Universal Robots PolyScope program: David.urp

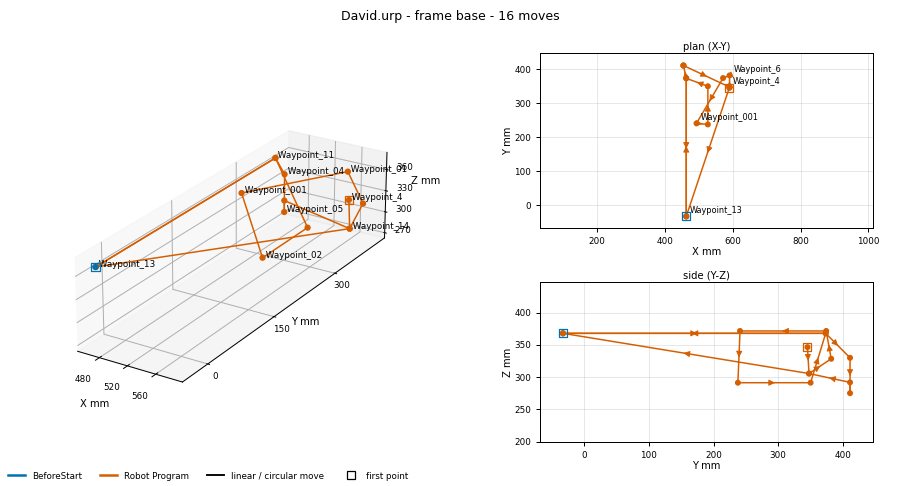
[picture p0: tool path of David.urp in frame base, 16 of 16 moves have a stored position in this frame; points joined in program order, loops and branches not executed]
Program David (installation=robINST_del2David directory=/programs/seminar/2526/zindovic_main createdIn=5.8.0.10253 lastSavedIn=5.8.0.10253 robotSerialNumber=20185500087)
Calibrated DH parameters: a=[0.000137, -0.413209, -0.387078, 0.000078, -0.000004, 0]; d=[0.162361, 46.755621, 39.772032, -86.394282, 0.099723, 0.099655]; alpha=[1.570462, -0.002125, 0.000722, 1.570578, -1.570334, 0]; deltaTheta=[0, -0.236012, 6.679269, -0.160076, 0, 0]
BeforeStart
  MoveJ speed 60 deg/s, acceleration 80 deg/s^2 (useActiveTCP=true) feature=Base
    Waypoint Waypoint_13: TCP in base x=463.075 y=-33.119 z=367.768 mm, rx=-2.2445 ry=2.187 rz=-0.1467 rad; joints [15.1, -81.195, -93.203, -92.685, 85.56, 13.599] deg; TCP offset x=0 y=0 z=159.6 mm, rx=0 ry=0 rz=0 rad
  URCap Gripper Activate (Robotiq_Grippers, Robotiq Inc.) dataModel(ResetAndActivateKey=false)
  If not digital_in[4]
    Popup Message (haltProgram=false message=Postavi skatlo k zadnjemu senzorju :) inputType=Text)
    Loop While (checkContinuously=false) expression=not digital_in[4]
      'prazen loop ne laufa :)'
      Wait Sleep waitTime=0.01
  open_socket := socket_open("192.168.65.102",50000,"student")
  Loop While (checkContinuously=false) expression=not open_socket
    open_socket := socket_open("192.168.65.102",50000,"student")
Robot Program (runOnlyOnce=true)
  MoveL speed 250 mm/s, acceleration 1200 mm/s^2 (useActiveTCP=true) feature=Base
    Waypoint Waypoint_4: TCP in base x=590.057 y=345.4 z=346.405 mm, rx=-2.197 ry=2.2194 rz=-0.0403 rad; joints [42.083, -114.466, -57.559, -96.882, 88.554, 42.722] deg
    URCap Gripper (Robotiq_Grippers, Robotiq Inc.) dataModel(position=0.0, force=0.0, speed=0.0, positionInDouble=0.0, forceInDouble=0.0, speedInDouble=0.0, slaveIds=[2], blocking=true)
  If not digital_in[5]
    Set DigitalOutput pin=digital_out[5]; digitalValue=1
  Loop While (checkContinuously=false) expression=not digital_in[5]
    'cakam da se skatla pripelje'
    Wait Sleep waitTime=0.01
  Set DigitalOutput pin=digital_out[5]; digitalValue=0
  'tcp ip skatla prispela'
  If open_socket
    was_send := socket_send_string("PRISPELA","student")
    Loop While (checkContinuously=false) expression=not was_send
      was_send := socket_send_string("PRISPELA","student")
      Wait Sleep waitTime=0.01
    Wait Sleep waitTime=0.01
  MoveL speed 250 mm/s, acceleration 1200 mm/s^2 (useActiveTCP=true) feature=Base
    Waypoint Waypoint_14: TCP in base x=590.692 y=347.823 z=305.527 mm, rx=2.1728 ry=-2.1663 rz=0.0699 rad; joints [42.721, -117.719, -57.552, -98.812, 87.209, 42.72] deg
    'premik za prijem pokrova'
  Set DigitalOutput pin=digital_out[0]; digitalValue=1
  'vkopi napajanje za kljucavnico'
  Wait Sleep waitTime=1
  Set DigitalOutput pin=digital_out[0]; digitalValue=0
  URCap Gripper (Robotiq_Grippers, Robotiq Inc.) dataModel(position=100.0, force=28.0, speed=0.0, positionInDouble=100.0, forceInDouble=28.0, speedInDouble=0.0, slaveIds=[2], blocking=true)
  'gripper primer pokrov'
  'tcp ip skatla odklenjena'
  If open_socket
    was_send := socket_send_string("ODKLENJENA","student")
    Loop While (checkContinuously=false) expression=not was_send
      was_send := socket_send_string("ODKLENJENA","student")
      Wait Sleep waitTime=0.01
    Wait Sleep waitTime=0.01
  SuppressedNode
    MoveL speed 250 mm/s, acceleration 1200 mm/s^2 (useActiveTCP=true) feature=Base
      Waypoint Waypoint_5: motionParameters(blendRadius=0.01); TCP in base x=590.703 y=347.825 z=305.52 mm, rx=2.1728 ry=-2.1663 rz=0.0699 rad; joints [42.721, -117.719, -57.554, -98.808, 87.207, 42.72] deg
      'dvigne pokrov'
  'tcp_ip skatla je odprta'
  If open_socket
    was_send := socket_send_string("ODPRTA","student")
    Loop While (checkContinuously=false) expression=not was_send
      was_send := socket_send_string("ODPRTA","student")
      Wait Sleep waitTime=0.01
    Wait Sleep waitTime=0.01
  'izklopi napajanje kljucavice (<4s)'
  MoveL speed 250 mm/s, acceleration 1200 mm/s^2 (useActiveTCP=true) feature=Base
    Waypoint Waypoint_6: TCP in base x=590.703 y=382.183 z=328.36 mm, rx=1.95 ry=-1.9516 rz=0.45 rad; joints [49.875, -136.415, -22.457, -133.186, 73.792, 53.142] deg; TCP offset x=0 y=0 z=159.6 mm, rx=0 ry=0 rz=0 rad
    'pokrov premakne blizje zadnjemu delu skatle'
  URCap Gripper (Robotiq_Grippers, Robotiq Inc.) dataModel(position=0.0, force=2.0, speed=100.0, positionInDouble=0.0, forceInDouble=2.0, speedInDouble=100.0, slaveIds=[2], blocking=true)
  'odpre prijemalo'
  MoveL speed 250 mm/s, acceleration 1200 mm/s^2 (useActiveTCP=true) feature=Base
    Waypoint Waypoint_01: TCP in base x=571.574 y=374.398 z=371.422 mm, rx=1.9617 ry=-2.392 rz=0.0295 rad; joints [44.751, -118.567, -46.705, -107.595, 89.15, 56.123] deg; TCP offset x=0 y=0 z=159.6 mm, rx=0 ry=0 rz=0 rad
    'se umakne za potisk pokrova'
  MoveL speed 250 mm/s, acceleration 1200 mm/s^2 (useActiveTCP=true) feature=Base
    Waypoint Waypoint_001: TCP in base x=493.333 y=240.994 z=371.405 mm, rx=1.9617 ry=-2.3919 rz=0.0295 rad; joints [40.5, -97.502, -74.971, -100.327, 88.983, 51.902] deg
    'vmesen korak za potisk pokrova'
  MoveL speed 250 mm/s, acceleration 1200 mm/s^2 (useActiveTCP=true) feature=Base
    Waypoint Waypoint_02: TCP in base x=526.745 y=237.719 z=291.293 mm, rx=1.9502 ry=-2.4581 rz=0.0124 rad; joints [37.744, -99.751, -84.689, -85.8, 89.558, 50.985] deg
    'se pripravi za potisk pokrova'
  MoveL speed 250 mm/s, acceleration 1200 mm/s^2 (useActiveTCP=true) feature=Base
    Waypoint Waypoint_03: TCP in base x=526.752 y=350.284 z=291.328 mm, rx=1.9502 ry=-2.4582 rz=0.0123 rad; joints [45.887, -107.465, -74.981, -87.85, 89.582, 59.122] deg
    'potisne pokrov'
  MoveL speed 250 mm/s, acceleration 1200 mm/s^2 (useActiveTCP=true) feature=Base
    Waypoint Waypoint_11: TCP in base x=463.07 y=373.635 z=367.778 mm, rx=-2.5524 ry=1.7928 rz=-0.1431 rad; joints [54.112, -100.735, -72.837, -95.286, 84.769, 34.317] deg
    'stran od skatle'
    Waypoint Waypoint_13: TCP in base x=463.075 y=-33.119 z=367.768 mm, rx=-2.2445 ry=2.187 rz=-0.1467 rad; joints [15.1, -81.195, -93.203, -92.685, 85.56, 13.599] deg
    'domov = opravi task'
    Wait Sleep waitTime=2
    Waypoint Waypoint_11: TCP in base x=463.07 y=373.635 z=367.778 mm, rx=-2.5524 ry=1.7928 rz=-0.1431 rad; joints [54.112, -100.735, -72.837, -95.286, 84.769, 34.317] deg
    'se postavi nad skatlo'
    URCap Gripper (Robotiq_Grippers, Robotiq Inc.) dataModel(position=0.0, force=2.0, speed=100.0, positionInDouble=0.0, forceInDouble=2.0, speedInDouble=100.0, slaveIds=[2], blocking=true)
    'odpre gripper'
    Waypoint Waypoint_04: TCP in base x=454.819 y=411.321 z=329.883 mm, rx=-2.3067 ry=2.1173 rz=-0.1463 rad; joints [56.923, -104.043, -73.887, -92.584, 84.659, 52.133] deg
    'premik nad pozicijo za pobiranje pokrova'
    Waypoint Waypoint_05: TCP in base x=454.826 y=411.326 z=275.129 mm, rx=-2.3067 ry=2.1173 rz=-0.1464 rad; joints [56.92, -104.296, -81.578, -84.644, 84.657, 52.136] deg
    'premik na pozicijo za pobiranje pokrova'
    URCap Gripper (Robotiq_Grippers, Robotiq Inc.) dataModel(position=100.0, force=30.0, speed=100.0, positionInDouble=100.0, forceInDouble=30.0, speedInDouble=100.0, slaveIds=[2], blocking=true)
    'zapre prijemalo'
    Waypoint Waypoint_06: TCP in base x=454.819 y=411.334 z=291.84 mm, rx=-2.3067 ry=2.1172 rz=-0.1463 rad; joints [56.921, -104.108, -79.367, -87.039, 84.659, 52.133] deg
    'dvigne pokrov'
    Waypoint Waypoint_14: TCP in base x=590.692 y=347.823 z=305.527 mm, rx=2.1728 ry=-2.1663 rz=0.0699 rad; joints [42.721, -117.719, -57.552, -98.812, 87.209, 42.72] deg
    'pokrov postavi v zacetno pozicijo'
    If open_socket
      was_send := socket_send_string("ZAPRTA","student")
      Loop While (checkContinuously=false) expression=not was_send
        was_send := socket_send_string("ZAPRTA","student")
        Wait Sleep waitTime=0.01
      Wait Sleep waitTime=0.01
    URCap Gripper (Robotiq_Grippers, Robotiq Inc.) dataModel(position=0.0, force=2.0, speed=100.0, positionInDouble=0.0, forceInDouble=2.0, speedInDouble=100.0, slaveIds=[2], blocking=true)
    'odpre gripper'
    Set DigitalOutput pin=digital_out[0]; digitalValue=1
    'vklopi napajanje za kljucavnico'
    Wait Sleep waitTime=1
    Set DigitalOutput pin=digital_out[0]; digitalValue=0
    'izklopi napajanje za kljucavnico'
    If open_socket
      was_send := socket_send_string("ZAKLENJENA","student")
      Loop While (checkContinuously=false) expression=not was_send
        was_send := socket_send_string("ZAKLENJENA","student")
        Wait Sleep waitTime=0.01
      Wait Sleep waitTime=0.01
    Waypoint Waypoint_13: TCP in base x=463.075 y=-33.119 z=367.768 mm, rx=-2.2445 ry=2.187 rz=-0.1467 rad; joints [15.1, -81.195, -93.203, -92.685, 85.56, 13.599] deg
    'domov'
  If digital_in[5]
    Set DigitalOutput pin=digital_out[5]; digitalValue=1
    'ce je skatla se pri senzorju posljemo naprej'
    'tcp_ip skatla sla naprej'
    If open_socket
      was_send := socket_send_string("ODPRAVLJENA","student")
      Loop While (checkContinuously=false) expression=not was_send
        was_send := socket_send_string("ODPRAVLJENA","student")
        Wait Sleep waitTime=0.01
      Wait Sleep waitTime=0.01
  Loop While (checkContinuously=false) expression=digital_in[5]
    'cakam da skatla ne bo vec pri senzorju'
  Set DigitalOutput pin=digital_out[5]; digitalValue=0
  Script: socket_close("student")
  Halt
